// TIA Portal project "汇博平台 - 副本_V15" (V15)

(* hardware
DEVICE "S7-1200 station_1"  S7-1200 Station
   slot 0: "Rack_0"  Rack  V1.0
   slot 1: "PLC_HostStation"  CPU 1215C DC/DC/DC  6ES7 215-1AG40-0XB0  V4.0
   slot 2: "DI 16x24VDC/DQ 16xRelay_1"  6ES7 223-1PL32-0XB0  V2.0
   slot 3: "DI 16x24VDC/DQ 16xRelay_2"  6ES7 223-1PL32-0XB0  V2.0
   slot 4: "DI 16x24VDC_1"  6ES7 221-1BH32-0XB0  V2.0
   slot 5: "DI 16x24VDC_2"  6ES7 221-1BH32-0XB0  V2.0
*)

// ===== PLC "PLC_HostStation"  CPU 1215C DC/DC/DC =====

VAR_GLOBAL   // PLC tag table "默认变量表"
   "System_Byte" AT %MB1 : Byte;
   "FirstScan" AT %M1.0 : Bool;
   "DiagStatusUpdate" AT %M1.1 : Bool;
   "AlwaysTRUE" AT %M1.2 : Bool;
   "AlwaysFALSE" AT %M1.3 : Bool;
   "Clock_Byte" AT %MB0 : Byte;
   "Clock_10Hz" AT %M0.0 : Bool;
   "Clock_5Hz" AT %M0.1 : Bool;
   "Clock_2.5Hz" AT %M0.2 : Bool;
   "Clock_2Hz" AT %M0.3 : Bool;
   "Clock_1.25Hz" AT %M0.4 : Bool;
   "Clock_1Hz" AT %M0.5 : Bool;
   "Clock_0.625Hz" AT %M0.6 : Bool;
   "Clock_0.5Hz" AT %M0.7 : Bool;
END_VAR

TYPE "Struct_WpState"
VERSION : 0.1
   STRUCT
      iNumName : Int;
      iWpType : Int;
      iMaterialQuality : Int;
      iCurrentState : Int;   // 0-无工件 1-毛坯 2-加工中 3-合格 4-不合格 5车完 6-铣完
   END_STRUCT;
END_TYPE

TYPE "Struct_RuningWpState"
VERSION : 0.1
   STRUCT
      RobotHandWpInfo : Array[1..2] of Int;
      LatChuckWpInfo : Int;
      CncChuckWpinfo : Int;
   END_STRUCT;
END_TYPE

DATA_BLOCK "DB_MesData"   // DB8
{ S7_Optimized_Access := 'FALSE' }
VERSION : 0.1
   VAR
      MesToPlc : Struct   // MES->PLC
         MesSendPlcCmd : Struct   // MES发给PLC的报文信息
            MesCmdCode : Int;   // MES命令码
            PickPos : Int;   // 取料位置
            PutPos : Int;   // 放料位置
            DeviceID : Int;   // 设备号（1=车床，2=加工中心）
            Reserve_3 : Int;   // 取料类型
            Reserve_4 : Int;   // 放料类型
            WpType : Int;   // 取料工件类型
            PutPosState : Int;   // 放料状态
            Reserve_1 : Int;   // 保留字
            Reserve_2 : Int;   // 保留字
         END_STRUCT;
         MesAckPlc_L : Struct   // MES响应PLC命令
            CmdAck : Int;   // 命令响应码
            StorePos : Int;   // 工件位置号
            Result : Int;   // 结果
            DeviceID : Int;   // 设备号（1=车床，2=加工中心）
            "--------Reserve_1" : Int;
         END_STRUCT;
         MesAckPlc_C : Struct   // MES响应PLC命令
            CmdAck : Int;   // 命令响应码
            StorePos : Int;   // 工件位置号
            Result : Int;   // 结果
            DeviceID : Int;   // 设备号（1=车床，2=加工中心）
            "--------Reserve_1" : Int;
         END_STRUCT;
      END_STRUCT;
      PlcToMes : Struct   // PLC-MES
         PlcSendMesCmd_L : Struct   // PLC 发给MES命令
            PlcCmdCode : Int;   // PLC命令码
            StorePos : Int;   // 工件位置号
            Result : Int;   // 执行结果
            DeviceID : Int;   // 设备号（1=车床，2=加工中心）
            "--------Reserve_1" : Int;
         END_STRUCT;
         PlcSendMesCmd_C : Struct   // PLC 发给MES命令
            PlcCmdCode : Int;   // PLC命令码
            StorePos : Int;   // 工件位置号
            Result : Int;   // 执行结果
            DeviceID : Int;   // 设备号（1=车床，2=加工中心）
            "--------Reserve_1" : Int;
         END_STRUCT;
         PlcAckMes : Struct   // PLC响应MES命令
            CmdAck : Int;   // PLC应答MES命令码
            PickPos : Int;   // 取料位
            PutPos : Int;   // 放料位
            DeviceID : Int;   // 设备号（1=车床，2=加工中心）
            "--------Reserve_1" : Int;
         END_STRUCT;
         PlcSendMesCmd_Rfid : Struct
            RfidAck : Int;   // 203 RFID全部写完成 204 RFID全部读完成（用户延时1S自己清除信号）
            Result : Int;   // 结果 1成功 2失败
            读取测量数据 : Int;   // 106 读取测量数据（用户延时1S自己清除信号）
            "--------Reserve_3" : Int;
            PLCstate : Int;
         END_STRUCT;
         RobotData : Struct
            RbtState : Int;   // 机器人当前状态 0停止 1故障 2运行中
            Home : Int;   // 机器人处于Home点
            mode : Int;   // 机器人当前模式
            RbtSpeed : Int;   // 机器人当前速度
            Axis1 : Int;   // 机器人轴1角度
            Axis2 : Int;   // 机器人轴2角度
            Axis3 : Int;   // 机器人轴3角度
            Axis4 : Int;   // 机器人轴4角度
            Axis5 : Int;   // 机器人轴5角度
            Axis6 : Int;   // 机器人轴6角度
            Axis7 : Int;   // 机器人轴7角度
            x : Int;   // 机器人X轴位置
            y : Int;   // 机器人Y轴位置
            z : Int;   // 机器人Z轴位置
            "a" : Int;   // 机器人a角度
            "b" : Int;   // 机器人b角度
            c : Int;   // 机器人c角度
         END_STRUCT;
         "-------Reserve_3" : Array[1..3] of Word;   // 保留字
      END_STRUCT;
      StoreWpExistInfo : Array[1..32] of Bool;   // 仓库工件信息
      Reserve : Array[1..3] of Word;   // 保留字
      LatAndCncState : Struct
         LatheDoorClose : Bool;
         LatheDoorOpen : Bool;
         LatheChuckState : Bool;
         ReserveBool_1 : Bool;
         ReserveBool_2 : Bool;
         ReserveBool_3 : Bool;
         ReserveBool_4 : Bool;
         ReserveBool_5 : Bool;
         ReserveWord_1 : Byte;
         CncDoorClose : Bool;   // 加工中心门关(0关闭 1打开）
         CncDoorOpen : Bool;   // 加工中心门开(0关闭 1打开）
         CncChuckState : Bool;   // 加工中心虎钳状态(0关闭 1打开）
         CncChuck2State : Bool;   // 加工中心零点夹具状态(0关闭 1打开）
         ReserveBool_7 : Bool;
         ReserveBool_8 : Bool;
         ReserveBool_9 : Bool;
         ReserveBool_10 : Bool;
         ReserveWord_2 : Byte;
      END_STRUCT;
      Reserve_1 : Array[1..3] of Word;   // 保留字
      StoreInfoDetail : Array[1..30] of "Struct_WpState";   // MES仓库信息
      机床采集数据 : Struct
         测量1数据整数 : Int;   // #600 整数部分，标定Z测头长度补偿，标定程序执行后#126的值，
         测量1数据小数 : Int;   // #600小数部分*1000
         测量2数据整数 : Int;   // #500 整数部分测头球半径补偿X
         测量2数据小数 : Int;   // #500小数部分*1000
         测量3数据整数 : Int;   // "#501 整数部分测头球半径补偿Y"
         测量3数据小数 : Int;   // #501小数部分*1000
         测量4数据整数 : Int;   // "#502 整数部分测头偏移补偿X"
         测量4数据小数 : Int;   // #502小数部分*1000
         测量5数据整数 : Int;   // "#503 整数部分测头偏移补偿Y"
         测量5数据小数 : Int;   // #503小数部分*1000
      END_STRUCT;
   END_VAR
BEGIN
END_DATA_BLOCK

DATA_BLOCK "SiemensHW_CONNECT"   // DB100
{ S7_Optimized_Access := 'TRUE' }
VERSION : 0.1
   VAR
      SiemensHW_RFID : IID_HW_CONNECT;
   END_VAR
BEGIN
END_DATA_BLOCK

ORGANIZATION_BLOCK "Main"   // OB1, LAD, ProgramCycle
TITLE = "Main Program Sweep (Cycle)"
{ S7_Optimized_Access := 'TRUE' }
VERSION : 0.1
   VAR_INPUT
      Initial_Call : Bool;   // Initial call of this OB
      Remanence : Bool;   // =True, if remanent data are available
   END_VAR
BEGIN
END_ORGANIZATION_BLOCK